SUBAPPLICATION Uebung_010 (* SoftKey_F1 auf DigitalOutput_Q1 *)
  (* Standard: 61499-2; Description: Copyright (c) 2023 Meisterschulen am Ostbahnhof This program and the accompanying materials are made available under the terms of the Eclipse Public License 2.0 which is available at https://www.eclipse.org/legal/epl-2.0/ SPDX-License-Identifier: EPL-2.0 *)
  (* Version 1.0, 2023-10-23, Franz Höpfinger, Meisterschulen am Ostbahnhof, initial API and implementation and/or initial documentation *)
  PACKAGE Uebungen;
  IMPORT Uebungen::const::UT::DefaultPool::SoftKey_F1;
  IMPORT logiBUS::io::DQ::logiBUS_DO::Output_Q1;
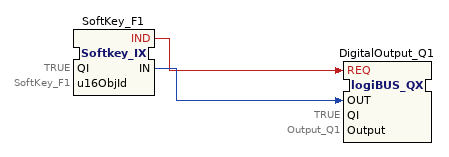
  FBS
    DigitalOutput_Q1 : logiBUS::io::DQ::logiBUS_QX(QI := TRUE, Output := Output_Q1);
    SoftKey_F1 : isobus::UT::io::Softkey::Softkey_IX(QI := TRUE, u16ObjId := SoftKey_F1);
  END_FBS
  EVENT_CONNECTIONS
    SoftKey_F1.IND TO DigitalOutput_Q1.REQ;
  END_CONNECTIONS
  DATA_CONNECTIONS
    SoftKey_F1.IN TO DigitalOutput_Q1.OUT;
  END_CONNECTIONS
END_SUBAPPLICATION
